FUNCTION_BLOCK Hysteresis_AR_AX (* Analog to Digital with Hysteresis *)
  (* Standard: 61499-2 *)
  (* Version 1.0, 2026-05-08, 4diac IDE *)
  PACKAGE logiBUS::signalprocessing::hysteresis;
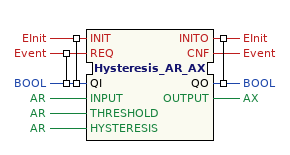
  EVENT_INPUT
    INIT : EInit WITH QI; (* Initialization Request *)
    REQ WITH QI; (* Normal Execution Request *)
  END_EVENT
  EVENT_OUTPUT
    INITO : EInit WITH QO; (* Initialization Confirm *)
    CNF; (* Execution Confirmation *)
  END_EVENT
  VAR_INPUT
    QI : BOOL; (* Input event qualifier *)
  END_VAR
  VAR_OUTPUT
    QO : BOOL;
  END_VAR
  SOCKETS
    INPUT : adapter::types::unidirectional::AR; (* Input value *)
    THRESHOLD : adapter::types::unidirectional::AR; (* Switch-off threshold *)
    HYSTERESIS : adapter::types::unidirectional::AR; (* Hysteresis band *)
  END_SOCKETS
  PLUGS
    OUTPUT : adapter::types::unidirectional::AX; (* Hysteresis output *)
  END_PLUGS
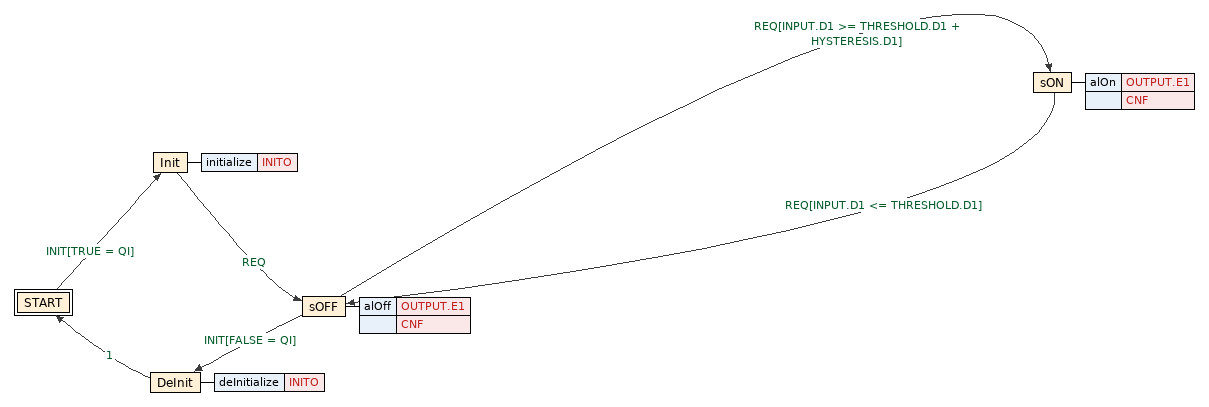
  EC_STATES
    START; (* Initial State *)
    Init : initialize -> INITO; (* Initialization *)
    sOFF : alOff -> OUTPUT.E1, -> CNF;
    DeInit : deInitialize -> INITO;
    sON : alOn -> OUTPUT.E1, -> CNF;
  END_STATES
  EC_TRANSITIONS
    START TO Init := INIT[TRUE = QI];
    Init TO sOFF := REQ;
    sOFF TO DeInit := INIT[FALSE = QI];
    sOFF TO sON := REQ[INPUT.D1 >= THRESHOLD.D1 + HYSTERESIS.D1];
    DeInit TO START := 1;
    sON TO sOFF := REQ[INPUT.D1 <= THRESHOLD.D1];
  END_TRANSITIONS
  ALGORITHM initialize IN ST:
QO := QI;
OUTPUT.D1 := BOOL#FALSE;
  END_ALGORITHM
  ALGORITHM deInitialize IN ST:
QO := BOOL#FALSE;
OUTPUT.D1 := BOOL#FALSE;
  END_ALGORITHM
  ALGORITHM alOff IN ST:
QO := QI;
OUTPUT.D1 := BOOL#FALSE;
  END_ALGORITHM
  ALGORITHM alOn IN ST:
QO := QI;
IF TRUE = QI THEN
	OUTPUT.D1 := BOOL#TRUE;
END_IF;
  END_ALGORITHM
END_FUNCTION_BLOCK
